TYPE E_AteqHandshake :
(
    CMD_IDLE,         	// No command active, ready for new command
    CMD_IN_PROGRESS,  	// ATEQ has acknowledged, command is running
	CMD_WAIT_CYCLE_END,
	CMD_EOC, 			// End Of Cycle
	CMD_DONE,
    CMD_ERROR,        	// Command completed with an error from ATEQ
    CMD_TIMEOUT,      	// Command did not complete within expected time
    CMD_RESET   
);
END_TYPE

(* stored: Version 1.1.0.1, ProductVersion 3.1.4024.15
   DUT E_AteqHandshake: Id {156ee2bd-c863-40c9-9647-6f25eaa354f0} *)
